FUNCTION_BLOCK TransferConveyor
VAR_INPUT
END_VAR
VAR_OUTPUT
END_VAR
VAR
	TransferConveyorToken : INT;
	PalletSensorNegEdge: F_TRIG;
	LeftEntryPosEdge: R_TRIG;
	RightEntryPosEdge: R_TRIG;
	
	PalletNegative : BOOL;
	LeftEntryPositive : BOOL;
	RightEntryPositive : BOOL;	


END_VAR

//If emergency button is activated or system isn't started or stopped, reset system token to 10.
IF NOT SystemStarted OR EmergencyActivated THEN
	TransferConveyorToken := 10;
END_IF
//Positive or negative edges of sensors.
PalletSensorNegEdge(CLK:= Pallet_Sensor, Q=> PalletNegative );
LeftEntryPosEdge(CLK:= At_Left_Entry , Q=> LeftEntryPositive );
RightEntryPosEdge(CLK:= At_Right_Entry , Q=> RightEntryPositive );
//Transfer conveyors working conditions.
CASE TransferConveyorToken OF
	//
	10:
		//Waiting for system start
		IF SystemStarted THEN
			TransferConveyorToken := 20;
		ELSE
			Transfer_Left := FALSE;
			Transfer_Right := FALSE;
		END_IF
	20:
		//Reset everything and wait for a new pallet.
		Load := FALSE;
		Transfer_Left := FALSE;
		Transfer_Right := FALSE;
		TransferringLeft := FALSE;
		TransferringRight := FALSE;
		
		IF Pallet_Sensor THEN
			TransferConveyorToken := 30;
		END_IF
	30:
		//Start loading conveyor until loaded sensor is activated. And decide where to transfer pallet according to low and high sensors.
		Load := TRUE;
		//
		IF Pallet_Sensor AND Low_Sensor AND NOT High_Sensor THEN
			TransferringLeft := TRUE;
		ELSIF Pallet_Sensor AND Low_Sensor AND High_Sensor THEN
			TransferringRight := TRUE;
		ELSIF PalletNegative THEN
			TransferBusy := TRUE;
		ELSIF Loaded AND TransferringLeft THEN
			TransferConveyorToken := 40;
		ELSIF Loaded AND TransferringRight THEN
			TransferConveyorToken := 50;
		END_IF
	
	40:
		//If the box is small, transfer it to left.
		Load := FALSE;
		Transfer_Left := TRUE;
		
		IF LeftEntryPositive THEN
			TransferBusy := FALSE;
			TransferConveyorToken := 10;
		END_IF
	
		
	50:
		//If the box is high, transfer it to right.
		Load := FALSE;
		Transfer_Right := TRUE;
		
		IF RightEntryPositive THEN
			TransferBusy := FALSE;
			TransferConveyorToken := 10;
		END_IF	
		
	ELSE
		//
		TransferConveyorToken := 10;
END_CASE

END_FUNCTION_BLOCK

(* stored: Version 1.1.0.1, ProductVersion 3.1.4024.6
   POU TransferConveyor: Id {d11d03f5-6453-43be-8072-36aeca7780e0}, SpecialFunc None *)
